FUNCTION FUN_GetSyncGroup_AllocationJob : Bool
VAR_INPUT
	Coordinates : ARRAY[0..3] OF st_Coordinate;
	NeedleInfo	:ARRAY[0..3] OF st_AllocatingNeedleInfo;
END_VAR

VAR_OUTPUT
	SyncGroup	:ARRAY[0..3] OF UINT ; 
END_VAR
VAR
	_SyncGroup	:ARRAY[0..3] OF UINT := [0,1,2,3];
	i : INT;
	j : INT;
END_VAR

FOR i:=0 TO 2 DO				
	FOR j:=i+1 TO 3 DO					
		IF Coordinates[i].X=Coordinates[j].X AND Coordinates[i].Y=Coordinates[j].Y  AND NeedleInfo[i].Station=NeedleInfo[j].Station THEN
			_SyncGroup[j] :=_SyncGroup[i];
		END_IF			
								
	END_FOR				
END_FOR			

SyncGroup:=_SyncGroup;

END_FUNCTION

(* stored: Version 1.1.0.1, ProductVersion 3.1.4024.13
   POU FUN_GetSyncGroup_AllocationJob: Id {8a0dc9df-2afc-4096-ba8f-7463002a6f7a}, SpecialFunc None *)
